(* PLC project Generated.project, CODESYS CODESYS V3.5 SP19 Patch 1 *)
(* stored: creationDateTime 2026-09-06T13:00:42.375521, modificationDateTime 2026-09-06T13:00:42.375521 *)

(* ======================================================================= 📊 FB_Diag_IhmHeartbeat — Surveillance bidirectionnelle Heartbeat IHM/PLC ─────────────────────────────────────────────────────────────── 🎯 Rôle : Surveillance toggle IHM, generation toggle PLC et diagnostic timeout 🛡️ Protection : FB de diagnostic autonome (sans action directe sur AU) 📄 Doc métier : DOC/AF/AF_Partie-12_Fonction_Diagnostic_v1.4.md ======================================================================= *)
FUNCTION_BLOCK FB_Diag_IhmHeartbeat
  VAR_INPUT
    Enable : BOOL;  (* === COMMANDES & REGLAGES === --> [CMD] Active la surveillance (FALSE = IHM invalide) *)
    TglHeartbeatIhm : BOOL;  (* --> [HW] Toggle IHM, inversion attendue toutes les 500 ms *)
    IhmTimeout : TIME := TIME#2s0ms;  (* --> [CFG] Absence maximale de front IHM *)
    PlcTogglePeriod : TIME := TIME#500ms;  (* --> [CFG] Periode du clignotant PLC *)
  END_VAR
  VAR_OUTPUT
    HeartbeatIhmOk : BOOL;  (* === ETATS & DIAGNOSTICS IHM === <-- [STAT] TRUE apres front IHM post-boot et avant timeout *)
    HeartbeatIhmTimeout : BOOL;  (* <-- [DIAG] TRUE = aucun front IHM depuis IhmTimeout *)
    TglHeartbeatPlc : BOOL;  (* <-- [STAT] Clignotant PLC a superviser cote IHM *)
    TimeSinceIhmEdge : TIME;  (* <-- [DIAG] Temps ecoule depuis le dernier front IHM *)
  END_VAR
  VAR
    IhmTimeoutTon : TON;  (* === SOUS-INSTANCES FB === * [INST] Timer de surveillance timeout IHM *)
    PlcToggleTon : TON;  (* * [INST] Timer clignotant heartbeat PLC *)
    LastIhmToggle : BOOL;  (* === CALCULS ET ETATS INTERNES === . [LOC] Memoire du dernier etat toggle IHM *)
    IhmEdgeSeen : BOOL;  (* . [LOC] Verrou front vu (interdit RETAIN au boot) *)
    IhmEdgeDetected : BOOL;  (* . [LOC] Front de changement toggle IHM detecte *)
  END_VAR

            

// === IMPLEMENTATION ===

{region "§1 Gate"}
// 🛑 Sans Enable, aucune valeur mémorisée ne peut déclarer l'IHM valide.
IF NOT Enable THEN
    HeartbeatIhmOk := FALSE;
    HeartbeatIhmTimeout := TRUE;
    TglHeartbeatPlc := FALSE;
    TimeSinceIhmEdge := T#0s;
    LastIhmToggle := TglHeartbeatIhm;
    IhmEdgeSeen := FALSE;
    IhmTimeoutTon(IN := FALSE, PT := IhmTimeout);
    PlcToggleTon(IN := FALSE, PT := PlcTogglePeriod);
    RETURN;
END_IF;
{endregion}

{region "§2 Front IHM"}
// 📥 Front par comparaison : l'IHM écrit un BOOL toggle, pas une impulsion courte.
IhmEdgeDetected := (TglHeartbeatIhm <> LastIhmToggle);
LastIhmToggle := TglHeartbeatIhm;
IF IhmEdgeDetected THEN
    IhmEdgeSeen := TRUE;
END_IF;
{endregion}

{region "§3 Timeout IHM"}
// ⏱️ Le timer repart à chaque front. Au boot, il atteint le timeout au bout de IhmTimeout.
// HeartbeatIhmOk reste TRUE tant que le timeout n'est pas expiré (boot propre sans alarme au scan 1).
IhmTimeoutTon(IN := NOT IhmEdgeDetected, PT := IhmTimeout);
TimeSinceIhmEdge := IhmTimeoutTon.ET;
HeartbeatIhmTimeout := IhmTimeoutTon.Q;
HeartbeatIhmOk := NOT HeartbeatIhmTimeout;
{endregion}

{region "§4 Clignotant PLC"}
// 💡 Clignotant PLC indépendant : information de vie pour l'IHM, jamais signal Signal Safety autonome.
PlcToggleTon(IN := NOT PlcToggleTon.Q, PT := PlcTogglePeriod);
IF PlcToggleTon.Q THEN
    TglHeartbeatPlc := NOT TglHeartbeatPlc;
END_IF;
{endregion}

          
END_FUNCTION_BLOCK
